FUNCTION_BLOCK FB_TestSomething EXTENDS FB_TestSuite
VAR_INPUT
END_VAR
VAR_OUTPUT
END_VAR
VAR
END_VAR

TestSum();
TestTrue();

METHOD TestTrue
VAR_INPUT
END_VAR
TEST('TestTrue');

AssertTrue(TRUE, 'Condition is not true');

TEST_FINISHED();
END_METHOD

METHOD TestSum
VAR_INPUT
END_VAR
TEST('TestSum');

AssertTrue(2+2=4, 'Condition is not true');

TEST_FINISHED();
END_METHOD

END_FUNCTION_BLOCK

(* stored: Version 1.1.0.1, ProductVersion 3.1.4024.12
   POU FB_TestSomething: Id {a5ea8811-5301-4f6c-aafd-b2e96e83b4a4}, SpecialFunc None
   Method TestTrue: Id {5dcda336-eb7c-4bc2-a049-4f178c78790e}
   Method TestSum: Id {976e0437-3cd7-4f7e-af64-671bf9c25b18} *)
